FUNCTION_BLOCK FB_Sensor_NC_TestDecorator EXTENDS FB_Sensor_TestParentDecorator 
VAR
	
END_VAR

(*			
	EVERDE sp. z o.o.
	Rafał Osajda		05.02.2025		TC 4026.13		wer. 0.0.0.1
	Zwraca aktualny stan czujnika
*)
METHOD IsActive : BOOL
IsActive			:= NOT THIS^.bContactTest;
END_METHOD

END_FUNCTION_BLOCK

(* stored: Version 1.1.0.1
   POU FB_Sensor_NC_TestDecorator: Id {98c11409-49db-4663-bbc7-0b96f80d8168}, SpecialFunc None
   Method IsActive: Id {96d392f8-0b42-4bef-b9b8-77dfed317f6f} *)
